// TwinCAT 3 PLC project Untitled1
// ProgramVersion: 3.1.4024.0
// libraries:
//   Tc2_Standard, * (Beckhoff Automation GmbH)
//   Tc2_System, * (Beckhoff Automation GmbH)
//   Tc3_EventLogger, * (Beckhoff Automation GmbH)
//   Tc3_Module, * (Beckhoff Automation GmbH)
// project tree:
//   DUTs/ T_MyType.TcDUT
//   / PlcTask.TcTTO
//   POUs/ FB_RPC.TcPOU, MAIN.TcPOU
// real-time tasks:
//   TASK PlcTask: cycle T#10ms, priority 20, ADS port 350

CONFIGURATION Untitled1
    RESOURCE PLC ON TwinCAT3
        TASK PlcTask(INTERVAL := T#10ms, PRIORITY := 20);
        PROGRAM MAIN WITH PlcTask : MAIN;
    END_RESOURCE
END_CONFIGURATION

// ---- DUTs/T_MyType.TcDUT
TYPE T_MyType :
STRUCT
	a : UDINT;
	b : LREAL;
	c : STRING;
END_STRUCT
END_TYPE

// ---- POUs/MAIN.TcPOU
PROGRAM MAIN
VAR
	fb_rpc : FB_RPC;
END_VAR

END_PROGRAM

// ---- POUs/FB_RPC.TcPOU
FUNCTION_BLOCK FB_RPC
VAR_INPUT
END_VAR
VAR_OUTPUT
END_VAR
VAR
	callCntAddition : UINT;
	callCntReadString : UINT;
	callCntWriteString : UINT;
	callCntReadStruct : UINT;
	callCntWriteStruct : UINT;
	
	m_myType : T_MyType;
	
	fbMsg : FB_TcMessage;
END_VAR

{attribute 'TcRpcEnable':='1'}
METHOD Addition : UINT
VAR_INPUT
	val_a : UINT;
	val_b : UINT;
END_VAR
callCntAddition := callCntAddition + 1;
Addition := val_a + val_b;
END_METHOD

METHOD FB_init : BOOL
VAR_INPUT
	bInitRetains : BOOL; // if TRUE, the retain variables are initialized (warm start / cold start)
	bInCopyCode : BOOL;  // if TRUE, the instance afterwards gets moved into the copy code (online change)
END_VAR
fbMsg.CreateEx(TC_EVENTS.RpcEventClass.WriteString, 0);
END_METHOD

{attribute 'TcRpcEnable':='1'}
METHOD ReadString : STRING
VAR_INPUT
END_VAR
VAR
	s_string : STRING := 'ReadString: Current call count: ';
END_VAR
callCntReadString := callCntReadString +1;
ReadString := CONCAT(s_string, UDINT_TO_STRING(callCntReadString));
END_METHOD

{attribute 'TcRpcEnable':='1'}
METHOD ReadStruct : T_MyType
VAR_INPUT
END_VAR
VAR
	myType : T_MyType;
	s_string : STRING := 'ReadStuct() - ';
END_VAR
callCntReadStruct := callCntReadStruct + 1;
myType.a := callCntReadStruct;
myType.b := 1.0 / UINT_TO_LREAL(callCntReadStruct);
myType.c := CONCAT(s_string, UDINT_TO_STRING(callCntReadStruct));

ReadStruct := myType;
END_METHOD

{attribute 'TcRpcEnable':='1'}
METHOD WriteString
VAR_INPUT
	in : STRING;
END_VAR
callCntWriteString := callCntWriteString +1;
fbMsg.Send(0); 
//ADSLOGSTR(
//	msgCtrlMask := ADSLOG_MSGTYPE_WARN OR ADSLOG_MSGTYPE_LOG,
//	msgFmtStr := 'String received: %s',
//	strArg := in
//	);
END_METHOD

{attribute 'TcRpcEnable':='1'}
METHOD WriteStruct : UINT
VAR_INPUT
	in : T_MyType;
END_VAR
m_myType.a := in.a;
m_myType.b := in.b;
m_myType.c := in.c;
callCntWriteStruct := callCntWriteStruct + 1;
WriteStruct := callCntWriteStruct;
END_METHOD

END_FUNCTION_BLOCK
